// TIA Portal V18 export
DATA_BLOCK "PruebaReadWrite"   // DB1
{ S7_Optimized_Access := 'FALSE' }
VERSION : 0.1
// stored: AutoNumber true, DBAccessibleFromOPCUA true, DBAccessibleFromWebserver true, IsOnlyStoredInLoadMemory false, IsWriteProtectedInAS false
   VAR
      var1 : Int := 3;
      var2 : Real := 3.8;
      var3 : String := 'Prueba R/W TiaPortal';
   END_VAR
BEGIN
END_DATA_BLOCK
